FUNCTION Camera_Init : BOOL
VAR_IN_OUT
	Camera : Cognex_Camera;
END_VAR

Camera.AcquisitionControl.Acquistion_Trigger_Enable := TRUE;
Camera.CameraState := Camera_State.Idel;

END_FUNCTION

(* stored: Version 1.1.0.1, ProductVersion 3.1.4024.10
   POU Camera_Init: Id {a70b5ab6-a358-4ede-ad88-10f3494b78fb}, SpecialFunc None *)
